{attribute 'GeneratedUsingTerminal: EK1122-0000-0018'}
{attribute addProperty BoxType "EK1122-0000-0018"}
{attribute addProperty Id "Beckhoff_EP3xxxsub_EK1100EK1100_AB5A94672A_0001_EP3162_0002_0016EP3162_CC62AFB732A_0002_EP3162_1002_0017EP3162_3BC5483034A_0003_EP3174_0002_0016EP3174_9DDA7BAE48A_0004_EP3174_0002_0017EP3174_9DDA7BAE48A_0005_EP3174_0002_0018EP3174_0E4717A052A_0006_EP3174_0002_0019EP3174_0E4717A052A_0007_EP3174_0002_0020EP3174_0E4717A052A_0008_EP3174_0002_0021EP3174_0E4717A052A_0009_EP3174_0002_0022EP3174_0E4717A052A_0010_EP3174_0002_0023EP3174_0E4717A052A_0011_EP3174_0092_0016EP3174_0E4717A052A_0012_EP3182_1002_0017EP3182_AA81812532A_0013_EP3182_1002_0018EP3182_3BC5483034A_0014_EP3182_1002_0019EP3182_3BC5483034A_0015_EP3182_1002_0020EP3182_3BC5483034A_0016_EP3184_0002_0016EP3184_9DDA7BAE48A_0017_EP3184_0002_0017EP3184_0E4717A052A_0018_EP3184_0002_0018EP3184_0E4717A052A_0019_EP3184_0002_0019EP3184_0E4717A052A_0020_EP3184_0002_0020EP3184_0E4717A052A_0021_EP3184_0002_0021EP3184_0E4717A052A_0022_EP3184_0402_0016EP3184_0E4717A052A_0023_EP3184_0402_0017EP3184_0E4717A052A_0024_EP3184_0402_0018EP3184_0E4717A052A_0025_EP3184_1002_0016EP3184_9DDA7BAE48A_0026_EP3184_1002_0017EP3184_9DDA7BAE48A_0027_EP3184_1002_0018EP3184_0E4717A052A_0028_EP3184_1002_0019EP3184_0E4717A052A_0029_EP3184_1002_0020EP3184_0E4717A052A_0030_EP3184_1002_0021EP3184_0E4717A052A_0031_EP3204_0002_0017EP3204_7A00DD1E52A_0032_EP3204_0002_0018EP3204_7A00DD1E52A_0033_EP3204_0002_0019EP3204_7A00DD1E52A_0034_EP3204_0002_0020EP3204_7A00DD1E52A_0035_EP3204_0002_0021EP3204_BF0B7ECE48A_0036_EP3314_0002_0016EP3314_CE6B02DE52A_0037_EP3314_0002_0017EP3314_CE6B02DE52A_0038_EP3314_0002_0018EP3314_CE6B02DE52A_0039_EP3314_0002_0019EP3314_6BF23D5548A_0040_EP3314_0002_0020EP3314_6BF23D5548A_0041_EP3314_0002_0021EP3314_6BF23D5548A_0042_EP3351_2022_0016EP3351_162281E230A_0043_EP3356_0022_0016EP3356_BED8D8B728A_0044_EP3356_0022_0017EP3356_BED8D8B728A_0045_EP3356_0022_0022EP3356_BED8D8B728A_0046_EP3632_0001_0016EP3632_A04CBB5A86A_0047_EP3632_0001_0017EP3632_A04CBB5A86A_0048_EP3744_0041_0016EP3744_F454EBD870A_0049_EP3744_0041_0017EP3744_F454EBD870A_0050_EP3744_0041_0018EP3744_F454EBD870A_0051_EP3744_0041_0019EP3744_F454EBD870A_0052_EP3744_0041_0020EP3744_F454EBD870A_0053_EP3744_0041_0021EP3744_F454EBD870A_0054_EP3744_1041_0016EP3744_F454EBD870A_0055_EP3744_1041_0017EP3744_F454EBD870A_0056_EP3744_1041_0018EP3744_F454EBD870A_0057_EP3744_1041_0019EP3744_F454EBD870A_0058_EP3744_1041_0020EP3744_F454EBD870A_0059_EP3744_1041_0021EP3744_F454EBD870A_0060_EP3752_0000_0017EP3752_944EB99242A_0061_EP3752_0000_0018EP3752_944EB99242"}
{attribute addProperty CRC "2562485555"}
{attribute addProperty Size "3196"}
TYPE Beckhoff_EP3xxxEK1122_98BC6D33 EXTENDS EK1122_AB5A9467 :
STRUCT
	{attribute addProperty Name "Beckhoff_EP3xxxsub_EK1100"}
	{attribute addProperty PreviousPort "Beckhoff EP3xxxEK1122 : D"}
	Beckhoff_EP3xxxsub_EK1100 : EK1100_AB5A9467;
	{attribute addProperty Name "A_0001_EP3162_0002_0016"}
	{attribute addProperty PreviousPort "Beckhoff EP3xxxsub EK1100 : C"}
	A_0001_EP3162_0002_0016 : EP3162_CC62AFB7;
	{attribute addProperty Name "A_0002_EP3162_1002_0017"}
	{attribute addProperty PreviousPort "A_0001(EP3162-0002-0016) : B"}
	A_0002_EP3162_1002_0017 : EP3162_3BC54830;
	{attribute addProperty Name "A_0003_EP3174_0002_0016"}
	{attribute addProperty PreviousPort "A_0002(EP3162-1002-0017) : B"}
	A_0003_EP3174_0002_0016 : EP3174_9DDA7BAE;
	{attribute addProperty Name "A_0004_EP3174_0002_0017"}
	{attribute addProperty PreviousPort "A_0003(EP3174-0002-0016) : B"}
	A_0004_EP3174_0002_0017 : EP3174_9DDA7BAE;
	{attribute addProperty Name "A_0005_EP3174_0002_0018"}
	{attribute addProperty PreviousPort "A_0004(EP3174-0002-0017) : B"}
	A_0005_EP3174_0002_0018 : EP3174_0E4717A0;
	{attribute addProperty Name "A_0006_EP3174_0002_0019"}
	{attribute addProperty PreviousPort "A_0005(EP3174-0002-0018) : B"}
	A_0006_EP3174_0002_0019 : EP3174_0E4717A0;
	{attribute addProperty Name "A_0007_EP3174_0002_0020"}
	{attribute addProperty PreviousPort "A_0006(EP3174-0002-0019) : B"}
	A_0007_EP3174_0002_0020 : EP3174_0E4717A0;
	{attribute addProperty Name "A_0008_EP3174_0002_0021"}
	{attribute addProperty PreviousPort "A_0007(EP3174-0002-0020) : B"}
	A_0008_EP3174_0002_0021 : EP3174_0E4717A0;
	{attribute addProperty Name "A_0009_EP3174_0002_0022"}
	{attribute addProperty PreviousPort "A_0008(EP3174-0002-0021) : B"}
	A_0009_EP3174_0002_0022 : EP3174_0E4717A0;
	{attribute addProperty Name "A_0010_EP3174_0002_0023"}
	{attribute addProperty PreviousPort "A_0009(EP3174-0002-0022) : B"}
	A_0010_EP3174_0002_0023 : EP3174_0E4717A0;
	{attribute addProperty Name "A_0011_EP3174_0092_0016"}
	{attribute addProperty PreviousPort "A_0010(EP3174-0002-0023) : B"}
	A_0011_EP3174_0092_0016 : EP3174_0E4717A0;
	{attribute addProperty Name "A_0012_EP3182_1002_0017"}
	{attribute addProperty PreviousPort "A_0011(EP3174-0092-0016) : B"}
	A_0012_EP3182_1002_0017 : EP3182_AA818125;
	{attribute addProperty Name "A_0013_EP3182_1002_0018"}
	{attribute addProperty PreviousPort "A_0012(EP3182-1002-0017) : B"}
	A_0013_EP3182_1002_0018 : EP3182_3BC54830;
	{attribute addProperty Name "A_0014_EP3182_1002_0019"}
	{attribute addProperty PreviousPort "A_0013(EP3182-1002-0018) : B"}
	A_0014_EP3182_1002_0019 : EP3182_3BC54830;
	{attribute addProperty Name "A_0015_EP3182_1002_0020"}
	{attribute addProperty PreviousPort "A_0014(EP3182-1002-0019) : B"}
	A_0015_EP3182_1002_0020 : EP3182_3BC54830;
	{attribute addProperty Name "A_0016_EP3184_0002_0016"}
	{attribute addProperty PreviousPort "A_0015(EP3182-1002-0020) : B"}
	A_0016_EP3184_0002_0016 : EP3184_9DDA7BAE;
	{attribute addProperty Name "A_0017_EP3184_0002_0017"}
	{attribute addProperty PreviousPort "A_0016(EP3184-0002-0016) : B"}
	A_0017_EP3184_0002_0017 : EP3184_0E4717A0;
	{attribute addProperty Name "A_0018_EP3184_0002_0018"}
	{attribute addProperty PreviousPort "A_0017(EP3184-0002-0017) : B"}
	A_0018_EP3184_0002_0018 : EP3184_0E4717A0;
	{attribute addProperty Name "A_0019_EP3184_0002_0019"}
	{attribute addProperty PreviousPort "A_0018(EP3184-0002-0018) : B"}
	A_0019_EP3184_0002_0019 : EP3184_0E4717A0;
	{attribute addProperty Name "A_0020_EP3184_0002_0020"}
	{attribute addProperty PreviousPort "A_0019(EP3184-0002-0019) : B"}
	A_0020_EP3184_0002_0020 : EP3184_0E4717A0;
	{attribute addProperty Name "A_0021_EP3184_0002_0021"}
	{attribute addProperty PreviousPort "A_0020(EP3184-0002-0020) : B"}
	A_0021_EP3184_0002_0021 : EP3184_0E4717A0;
	{attribute addProperty Name "A_0022_EP3184_0402_0016"}
	{attribute addProperty PreviousPort "A_0021(EP3184-0002-0021) : B"}
	A_0022_EP3184_0402_0016 : EP3184_0E4717A0;
	{attribute addProperty Name "A_0023_EP3184_0402_0017"}
	{attribute addProperty PreviousPort "A_0022(EP3184-0402-0016) : B"}
	A_0023_EP3184_0402_0017 : EP3184_0E4717A0;
	{attribute addProperty Name "A_0024_EP3184_0402_0018"}
	{attribute addProperty PreviousPort "A_0023(EP3184-0402-0017) : B"}
	A_0024_EP3184_0402_0018 : EP3184_0E4717A0;
	{attribute addProperty Name "A_0025_EP3184_1002_0016"}
	{attribute addProperty PreviousPort "A_0024(EP3184-0402-0018) : B"}
	A_0025_EP3184_1002_0016 : EP3184_9DDA7BAE;
	{attribute addProperty Name "A_0026_EP3184_1002_0017"}
	{attribute addProperty PreviousPort "A_0025(EP3184-1002-0016) : B"}
	A_0026_EP3184_1002_0017 : EP3184_9DDA7BAE;
	{attribute addProperty Name "A_0027_EP3184_1002_0018"}
	{attribute addProperty PreviousPort "A_0026(EP3184-1002-0017) : B"}
	A_0027_EP3184_1002_0018 : EP3184_0E4717A0;
	{attribute addProperty Name "A_0028_EP3184_1002_0019"}
	{attribute addProperty PreviousPort "A_0027(EP3184-1002-0018) : B"}
	A_0028_EP3184_1002_0019 : EP3184_0E4717A0;
	{attribute addProperty Name "A_0029_EP3184_1002_0020"}
	{attribute addProperty PreviousPort "A_0028(EP3184-1002-0019) : B"}
	A_0029_EP3184_1002_0020 : EP3184_0E4717A0;
	{attribute addProperty Name "A_0030_EP3184_1002_0021"}
	{attribute addProperty PreviousPort "A_0029(EP3184-1002-0020) : B"}
	A_0030_EP3184_1002_0021 : EP3184_0E4717A0;
	{attribute addProperty Name "A_0031_EP3204_0002_0017"}
	{attribute addProperty PreviousPort "A_0030(EP3184-1002-0021) : B"}
	A_0031_EP3204_0002_0017 : EP3204_7A00DD1E;
	{attribute addProperty Name "A_0032_EP3204_0002_0018"}
	{attribute addProperty PreviousPort "A_0031(EP3204-0002-0017) : B"}
	A_0032_EP3204_0002_0018 : EP3204_7A00DD1E;
	{attribute addProperty Name "A_0033_EP3204_0002_0019"}
	{attribute addProperty PreviousPort "A_0032(EP3204-0002-0018) : B"}
	A_0033_EP3204_0002_0019 : EP3204_7A00DD1E;
	{attribute addProperty Name "A_0034_EP3204_0002_0020"}
	{attribute addProperty PreviousPort "A_0033(EP3204-0002-0019) : B"}
	A_0034_EP3204_0002_0020 : EP3204_7A00DD1E;
	{attribute addProperty Name "A_0035_EP3204_0002_0021"}
	{attribute addProperty PreviousPort "A_0034(EP3204-0002-0020) : B"}
	A_0035_EP3204_0002_0021 : EP3204_BF0B7ECE;
	{attribute addProperty Name "A_0036_EP3314_0002_0016"}
	{attribute addProperty PreviousPort "A_0035(EP3204-0002-0021) : B"}
	A_0036_EP3314_0002_0016 : EP3314_CE6B02DE;
	{attribute addProperty Name "A_0037_EP3314_0002_0017"}
	{attribute addProperty PreviousPort "A_0036(EP3314-0002-0016) : B"}
	A_0037_EP3314_0002_0017 : EP3314_CE6B02DE;
	{attribute addProperty Name "A_0038_EP3314_0002_0018"}
	{attribute addProperty PreviousPort "A_0037(EP3314-0002-0017) : B"}
	A_0038_EP3314_0002_0018 : EP3314_CE6B02DE;
	{attribute addProperty Name "A_0039_EP3314_0002_0019"}
	{attribute addProperty PreviousPort "A_0038(EP3314-0002-0018) : B"}
	A_0039_EP3314_0002_0019 : EP3314_6BF23D55;
	{attribute addProperty Name "A_0040_EP3314_0002_0020"}
	{attribute addProperty PreviousPort "A_0039(EP3314-0002-0019) : B"}
	A_0040_EP3314_0002_0020 : EP3314_6BF23D55;
	{attribute addProperty Name "A_0041_EP3314_0002_0021"}
	{attribute addProperty PreviousPort "A_0040(EP3314-0002-0020) : B"}
	A_0041_EP3314_0002_0021 : EP3314_6BF23D55;
	{attribute addProperty Name "A_0042_EP3351_2022_0016"}
	{attribute addProperty PreviousPort "A_0041(EP3314-0002-0021) : B"}
	A_0042_EP3351_2022_0016 : EP3351_162281E2;
	{attribute addProperty Name "A_0043_EP3356_0022_0016"}
	{attribute addProperty PreviousPort "A_0042(EP3351-2022-0016) : B"}
	A_0043_EP3356_0022_0016 : EP3356_BED8D8B7;
	{attribute addProperty Name "A_0044_EP3356_0022_0017"}
	{attribute addProperty PreviousPort "A_0043(EP3356-0022-0016) : B"}
	A_0044_EP3356_0022_0017 : EP3356_BED8D8B7;
	{attribute addProperty Name "A_0045_EP3356_0022_0022"}
	{attribute addProperty PreviousPort "A_0044(EP3356-0022-0017) : B"}
	A_0045_EP3356_0022_0022 : EP3356_BED8D8B7;
	{attribute addProperty Name "A_0046_EP3632_0001_0016"}
	{attribute addProperty PreviousPort "A_0045(EP3356-0022-0022) : B"}
	A_0046_EP3632_0001_0016 : EP3632_A04CBB5A;
	{attribute addProperty Name "A_0047_EP3632_0001_0017"}
	{attribute addProperty PreviousPort "A_0046(EP3632-0001-0016) : B"}
	A_0047_EP3632_0001_0017 : EP3632_A04CBB5A;
	{attribute addProperty Name "A_0048_EP3744_0041_0016"}
	{attribute addProperty PreviousPort "A_0047(EP3632-0001-0017) : B"}
	A_0048_EP3744_0041_0016 : EP3744_F454EBD8;
	{attribute addProperty Name "A_0049_EP3744_0041_0017"}
	{attribute addProperty PreviousPort "A_0048(EP3744-0041-0016) : B"}
	A_0049_EP3744_0041_0017 : EP3744_F454EBD8;
	{attribute addProperty Name "A_0050_EP3744_0041_0018"}
	{attribute addProperty PreviousPort "A_0049(EP3744-0041-0017) : B"}
	A_0050_EP3744_0041_0018 : EP3744_F454EBD8;
	{attribute addProperty Name "A_0051_EP3744_0041_0019"}
	{attribute addProperty PreviousPort "A_0050(EP3744-0041-0018) : B"}
	A_0051_EP3744_0041_0019 : EP3744_F454EBD8;
	{attribute addProperty Name "A_0052_EP3744_0041_0020"}
	{attribute addProperty PreviousPort "A_0051(EP3744-0041-0019) : B"}
	A_0052_EP3744_0041_0020 : EP3744_F454EBD8;
	{attribute addProperty Name "A_0053_EP3744_0041_0021"}
	{attribute addProperty PreviousPort "A_0052(EP3744-0041-0020) : B"}
	A_0053_EP3744_0041_0021 : EP3744_F454EBD8;
	{attribute addProperty Name "A_0054_EP3744_1041_0016"}
	{attribute addProperty PreviousPort "A_0053(EP3744-0041-0021) : B"}
	A_0054_EP3744_1041_0016 : EP3744_F454EBD8;
	{attribute addProperty Name "A_0055_EP3744_1041_0017"}
	{attribute addProperty PreviousPort "A_0054(EP3744-1041-0016) : B"}
	A_0055_EP3744_1041_0017 : EP3744_F454EBD8;
	{attribute addProperty Name "A_0056_EP3744_1041_0018"}
	{attribute addProperty PreviousPort "A_0055(EP3744-1041-0017) : B"}
	A_0056_EP3744_1041_0018 : EP3744_F454EBD8;
	{attribute addProperty Name "A_0057_EP3744_1041_0019"}
	{attribute addProperty PreviousPort "A_0056(EP3744-1041-0018) : B"}
	A_0057_EP3744_1041_0019 : EP3744_F454EBD8;
	{attribute addProperty Name "A_0058_EP3744_1041_0020"}
	{attribute addProperty PreviousPort "A_0057(EP3744-1041-0019) : B"}
	A_0058_EP3744_1041_0020 : EP3744_F454EBD8;
	{attribute addProperty Name "A_0059_EP3744_1041_0021"}
	{attribute addProperty PreviousPort "A_0058(EP3744-1041-0020) : B"}
	A_0059_EP3744_1041_0021 : EP3744_F454EBD8;
	{attribute addProperty Name "A_0060_EP3752_0000_0017"}
	{attribute addProperty PreviousPort "A_0059(EP3744-1041-0021) : B"}
	A_0060_EP3752_0000_0017 : EP3752_944EB992;
	{attribute addProperty Name "A_0061_EP3752_0000_0018"}
	{attribute addProperty PreviousPort "A_0060(EP3752-0000-0017) : B"}
	A_0061_EP3752_0000_0018 : EP3752_944EB992;
END_STRUCT
END_TYPE

(* stored: Version 1.2.0.0, ProductVersion 3.1.4024.9
   DUT Beckhoff_EP3xxxEK1122_98BC6D33: Id {dfe2b609-65fa-4c98-a6f1-cd488679be25} *)
